// TIA Portal project "LabKlipovi" (V14)

(* hardware
DEVICE "S71500/ET200MP station_1"  S7-1500 station
   slot 0: "Rail_0"  Rack  6ES7 590-1***0-0AA0
   slot 1: "PLC_1"  CPU 1511-1 PN  6ES7 511-1AK00-0AB0  V1.0
      slot 3: "CPU display_1"  6ES7591-1XA00-0AA0
   slot 2: "DI 16x24VDC HF_1"  DI 16x24VDC HF  6ES7 521-1BH00-0AB0  V1.0
   slot 3: "DQ 16x24VDC/0.5A ST_1"  DQ 16x24VDC/0.5A ST  6ES7 522-1BH00-0AB0  V1.0
   slot 4: "AI 8xU/I/RTD/TC ST_1"  AI 8xU/I/RTD/TC ST  6ES7 531-7KF00-0AB0  V2.0
*)

// ===== PLC "PLC_1"  CPU 1511-1 PN =====

VAR_GLOBAL   // PLC tag table "Tag table_1"
   "K1L" AT %I0.0 : Bool;
   "K1D" AT %I0.1 : Bool;
   "K2L" AT %I0.2 : Bool;
   "K2D" AT %I0.3 : Bool;
   "K3L" AT %I0.4 : Bool;
   "K3D" AT %I0.5 : Bool;
   "K4L" AT %I0.6 : Bool;
   "K4D" AT %I0.7 : Bool;
   "Komanda_K1L" AT %Q0.0 : Bool;
   "Komanda_K1D" AT %Q0.1 : Bool;
   "Komanda_K2L" AT %Q0.2 : Bool;
   "Komanda_K2D" AT %Q0.3 : Bool;
   "Komanda_K3L" AT %Q0.4 : Bool;
   "Komanda_K4L" AT %Q0.6 : Bool;
   "K1_AN" AT %IW2 : Int;
   "K4_AN" AT %IW4 : Int;
   "Timer_12s" AT %T0 : Timer;
   "Counter_0" AT %C0 : Counter;
   "Timer_9s" AT %T1 : Timer;
   "Crank" AT %M0.0 : Bool;
END_VAR

DATA_BLOCK "Block_1_DB"   // DB1
{ S7_Optimized_Access := 'TRUE' }
VERSION : 0.1
// stored: InstanceOfName Block_1
"Block_1"
BEGIN
END_DATA_BLOCK

FUNCTION_BLOCK "Block_1"   // FB1, GRAPH_PLUS
{ S7_Optimized_Access := 'TRUE' }
VERSION : 0.1
   VAR_INPUT
      OFF_SQ : Bool := false;   // Turn sequence off
      INIT_SQ : Bool := false;   // Set sequence to initial state
      ACK_EF : Bool := false;   // Acknowledge all errors and faults
      S_PREV : Bool := false;   // Output previous step in parameter S_NO
      S_NEXT : Bool := false;   // Indicate next step in parameter S_NO
      SW_AUTO : Bool := false;   // Automatic mode
      SW_TAP : Bool := false;   // Semiautomatic/switch with transition
      SW_TOP : Bool := false;   // Semiautomatic/ignore transition
      SW_MAN : Bool := false;   // Manual mode
      S_SEL : Int := 0;   // Select step to be output to S_NO
      S_ON : Bool := false;   // Activate step indicated in S_NO
      S_OFF : Bool := false;   // Deactivate step indicated S_NO
      T_PUSH : Bool := false;   // Enable transition to switch in semi automatic mode
   END_VAR
   VAR_OUTPUT
      S_NO : Int := 0;   // Step number
      S_MORE : Bool := false;   // More steps are available and can be shown in S_NO
      S_ACTIVE : Bool := false;   // Step indicated in S_NO is active
      ERR_FLT : Bool := false;   // Interlock or supervision group error
      AUTO_ON : Bool := false;   // Automatic mode is active
      TAP_ON : Bool := false;   // Semiautomatic mode/step with transition enabled
      TOP_ON : Bool := false;   // Semiautomatic mode/ignore transition enabled
      MAN_ON : Bool := false;   // Manual mode is active
   END_VAR
   VAR
      HMI_INFO : Array[0..10] of UInt;
      IF_PAR : G7_IfParPlus_V2;
      RT_DATA : G7_RTDataPlus_V2;   // Internal data area
      Trans1 : G7_TransitionPlus_V2;   // Transition structure
      Trans2 : G7_TransitionPlus_V2;   // Transition structure
      Trans3 : G7_TransitionPlus_V2;   // Transition structure
      Trans4 : G7_TransitionPlus_V2;   // Transition structure
      Trans5 : G7_TransitionPlus_V2;   // Transition structure
      Trans7 : G7_TransitionPlus_V2;   // Transition structure
      Trans8 : G7_TransitionPlus_V2;   // Transition structure
      Trans10 : G7_TransitionPlus_V2;   // Transition structure
      Trans11 : G7_TransitionPlus_V2;   // Transition structure
      Trans12 : G7_TransitionPlus_V2;   // Transition structure
      Trans14 : G7_TransitionPlus_V2;   // Transition structure
      Trans15 : G7_TransitionPlus_V2;   // Transition structure
      Trans16 : G7_TransitionPlus_V2;   // Transition structure
      Trans17 : G7_TransitionPlus_V2;   // Transition structure
      Trans18 : G7_TransitionPlus_V2;   // Transition structure
      Trans19 : G7_TransitionPlus_V2;   // Transition structure
      Init : G7_StepPlus_V2;   // Step structure
      Step2 : G7_StepPlus_V2;   // Step structure
      Step3 : G7_StepPlus_V2;   // Step structure
      Step4 : G7_StepPlus_V2;   // Step structure
      Step5 : G7_StepPlus_V2;   // Step structure
      Step7 : G7_StepPlus_V2;   // Step structure
      Step8 : G7_StepPlus_V2;   // Step structure
      Step10 : G7_StepPlus_V2;   // Step structure
      Step11 : G7_StepPlus_V2;   // Step structure
      Step12 : G7_StepPlus_V2;   // Step structure
      Step13 : G7_StepPlus_V2;   // Step structure
      Step14 : G7_StepPlus_V2;   // Step structure
      Step15 : G7_StepPlus_V2;   // Step structure
      Step16 : G7_StepPlus_V2;   // Step structure
      Step17 : G7_StepPlus_V2;   // Step structure
      SINI : Array[0..3] of USInt;
      LSTT : Array[0..15] of USInt;
      ATAJ : Array[0..15] of USInt;
      ATAB : Array[0..15] of USInt;
      PSTT : Array[0..15] of USInt;
      NSTT : Array[0..15] of USInt;
      ASSJ : Array[0..14] of USInt;
      ASSB : Array[0..14] of USInt;
      PTTS : Array[0..14] of USInt;
      NTTS : Array[0..14] of USInt;
      SW_SQTS : Array[0..14] of USInt;
      SWITCH : Array[0..1] of USInt;
      TVX : Array[0..5] of USInt;
      TTX : Array[0..5] of USInt;
      TSX : Array[0..3] of USInt;
      S00X : Array[0..3] of USInt;
      SOFFX : Array[0..3] of USInt;
      SONX : Array[0..3] of USInt;
      SAX : Array[0..3] of USInt;
      SERRX : Array[0..15] of USInt;
      SMX : Array[0..15] of USInt;
      S0X : Array[0..15] of USInt;
      S1X : Array[0..15] of USInt;
      IL_ALARM_INST : Program_Alarm;
      SUP_ALARM_INST : Program_Alarm;
      STEP_TIME_ALARM_INST : Program_Alarm;
      IEC_TIMER_INST : IEC_TIMER;
   END_VAR
   // SINI[0] := 2;
   // LSTT[0] := 255;
   // LSTT[1] := 255;
   // LSTT[2] := 255;
   // LSTT[3] := 255;
   // LSTT[4] := 255;
   // LSTT[5] := 255;
   // ATAJ[1] := 1;
   // ATAJ[2] := 2;
   // ATAJ[3] := 3;
   // ATAJ[4] := 4;
   // ATAJ[5] := 5;
   // ATAB[1] := 1;
   // ATAB[2] := 2;
   // ATAB[3] := 3;
   // ATAB[4] := 4;
   // ATAB[5] := 5;
   // PSTT[1] := 1;
   // PSTT[2] := 2;
   // PSTT[3] := 3;
   // PSTT[4] := 4;
   // PSTT[5] := 5;
   // NSTT[0] := 1;
   // NSTT[1] := 2;
   // NSTT[2] := 3;
   // NSTT[3] := 4;
   // NSTT[4] := 5;
   // NSTT[5] := 6;
   // ASSJ[1] := 1;
   // ASSJ[2] := 2;
   // ASSJ[3] := 3;
   // ASSJ[4] := 4;
   // ASSJ[5] := 5;
   // ASSB[1] := 1;
   // ASSB[2] := 2;
   // ASSB[3] := 3;
   // ASSB[4] := 4;
   // ASSB[5] := 7;
   // PTTS[0] := 255;
   // PTTS[2] := 1;
   // PTTS[3] := 2;
   // PTTS[4] := 3;
   // PTTS[5] := 4;
   // NTTS[1] := 1;
   // NTTS[2] := 2;
   // NTTS[3] := 3;
   // NTTS[4] := 4;
   // NTTS[5] := 5;
   // TVX[0] := 16#1;
   // TTX[0] := 16#1;
   // TSX[0] := 16#1;
   // S00X[0] := 16#1;
   // SOFFX[0] := 16#1;
   // SONX[0] := 16#1;
   // SAX[0] := 16#1;
   // SERRX[0] := 16#1;
   // SMX[0] := 16#1;
   // S0X[0] := 16#1;
   // S1X[0] := 16#1;
   // NTTS[8] := 8;
   // PTTS[8] := 7;
   // ASSB[8] := 8;
   // SW_SQTS[8] := 2;
   // ASSJ[8] := 8;
   // SINI[2] := 255;
   // SINI[3] := 255;
   // LSTT[6] := 5;
   // LSTT[7] := 255;
   // NSTT[8] := 9;
   // ATAJ[6] := 6;
   // ATAJ[7] := 7;
   // PSTT[8] := 8;
   // ATAB[6] := 6;
   // ATAB[7] := 7;
   // ATAB[8] := 8;
   // PSTT[6] := 6;
   // PSTT[7] := 7;
   // ATAJ[8] := 8;
   // NSTT[6] := 5;
   // NSTT[7] := 8;
   // LSTT[8] := 255;
   // ASSJ[6] := 6;
   // ASSJ[7] := 7;
   // ASSB[6] := 6;
   // ASSB[7] := 5;
   // PTTS[6] := 5;
   // PTTS[7] := 4;
   // NTTS[6] := 6;
   // NTTS[7] := 7;
   // SW_SQTS[5] := 1;
   // SW_SQTS[6] := 1;
   // SW_SQTS[7] := 2;
   // SWITCH[0] := 192;
   // LSTT[11] := 255;
   // LSTT[9] := 255;
   // LSTT[10] := 3;
   // ATAJ[9] := 9;
   // ATAJ[10] := 10;
   // ATAB[9] := 10;
   // ATAB[10] := 9;
   // PSTT[9] := 10;
   // PSTT[10] := 10;
   // NSTT[9] := 11;
   // NSTT[10] := 3;
   // ASSJ[9] := 9;
   // ASSB[9] := 9;
   // PTTS[9] := 8;
   // NTTS[9] := 11;
   // SW_SQTS[9] := 2;
   // ATAJ[11] := 11;
   // ATAB[11] := 11;
   // PSTT[11] := 9;
   // NSTT[11] := 10;
   // ASSJ[10] := 10;
   // ASSB[10] := 10;
   // PTTS[10] := 11;
   // NTTS[10] := 9;
   // SW_SQTS[10] := 2;
   // LSTT[12] := 255;
   // LSTT[13] := 255;
   // LSTT[14] := 255;
   // LSTT[15] := 255;
   // ATAJ[12] := 12;
   // ATAJ[13] := 13;
   // ATAJ[14] := 14;
   // ATAJ[15] := 15;
   // ATAB[12] := 12;
   // ATAB[13] := 13;
   // ATAB[14] := 14;
   // ATAB[15] := 15;
   // PSTT[12] := 11;
   // PSTT[13] := 12;
   // PSTT[14] := 13;
   // PSTT[15] := 14;
   // NSTT[12] := 12;
   // NSTT[13] := 13;
   // NSTT[14] := 14;
   // NSTT[15] := 255;
   // ASSJ[11] := 11;
   // ASSJ[12] := 12;
   // ASSJ[13] := 13;
   // ASSJ[14] := 14;
   // ASSB[11] := 11;
   // ASSB[12] := 12;
   // ASSB[13] := 13;
   // ASSB[14] := 14;
   // PTTS[11] := 9;
   // PTTS[12] := 12;
   // PTTS[13] := 13;
   // PTTS[14] := 14;
   // NTTS[11] := 12;
   // NTTS[12] := 13;
   // NTTS[13] := 14;
   // NTTS[14] := 15;
   // SW_SQTS[11] := 3;
   // SW_SQTS[12] := 3;
   // SW_SQTS[13] := 3;
   // SW_SQTS[14] := 3;
   // SWITCH[1] := 34;
BEGIN
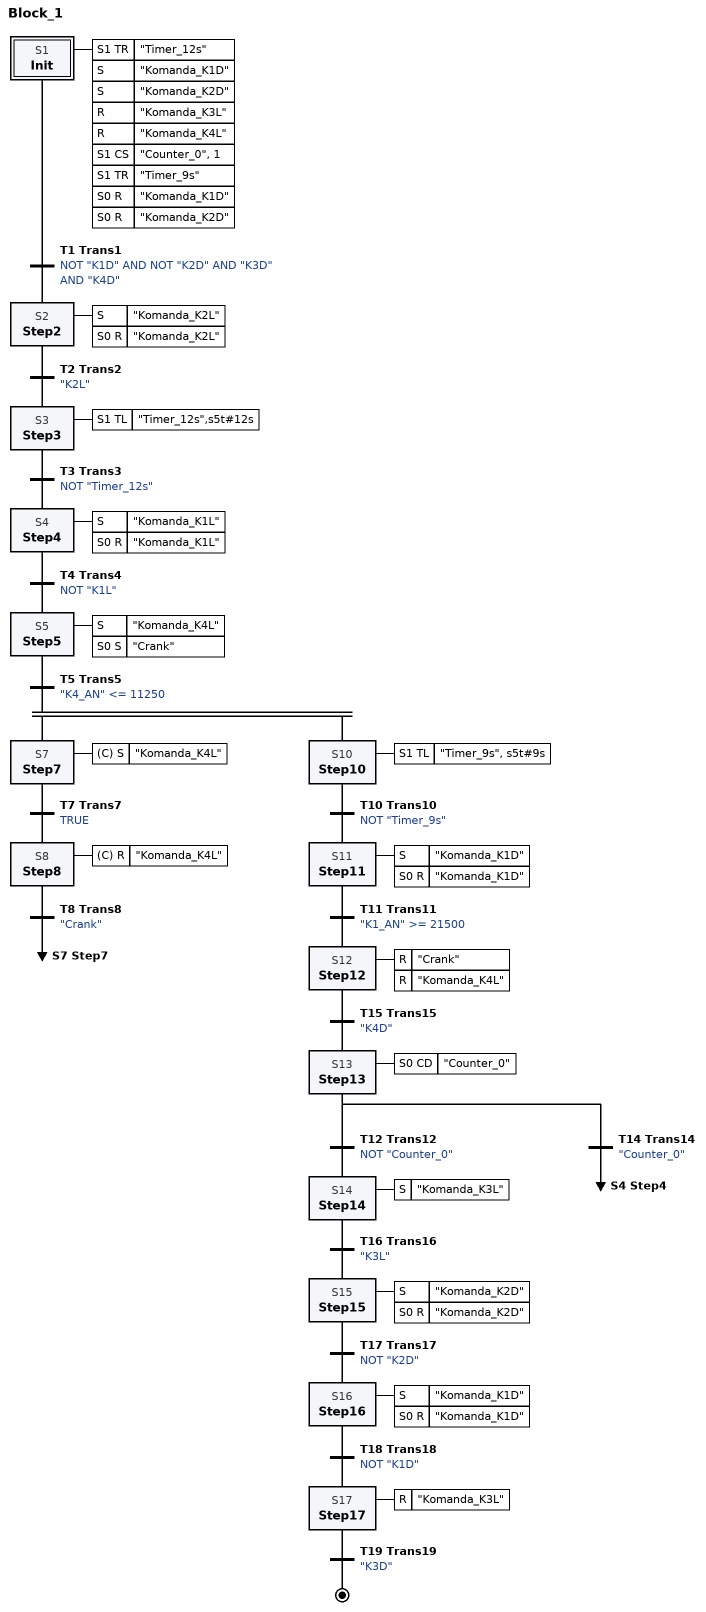
   // sequencer 1
   INITIAL_STEP Init:   // S1, max time T#10S, warning time T#7S
          S1  TR   "Timer_12s"
              S    "Komanda_K1D"
              S    "Komanda_K2D"
              R    "Komanda_K3L"
              R    "Komanda_K4L"
          S1  CS   "Counter_0", 1
          S1  TR   "Timer_9s"
          S0  R    "Komanda_K1D"
          S0  R    "Komanda_K2D"
   END_STEP
   TRANSITION Trans1 FROM Init TO Step2   // T1
      := NOT "K1D" AND NOT "K2D" AND "K3D" AND "K4D";
   END_TRANSITION
   STEP Step2:   // S2, max time T#10S, warning time T#7S
              S    "Komanda_K2L"
          S0  R    "Komanda_K2L"
   END_STEP
   TRANSITION Trans2 FROM Step2 TO Step3   // T2
      := "K2L";
   END_TRANSITION
   STEP Step3:   // S3, max time T#10S, warning time T#7S
          S1  TL   "Timer_12s",s5t#12s
   END_STEP
   TRANSITION Trans3 FROM Step3 TO Step4   // T3
      := NOT "Timer_12s";
   END_TRANSITION
   STEP Step4:   // S4, max time T#10S, warning time T#7S
              S    "Komanda_K1L"
          S0  R    "Komanda_K1L"
   END_STEP
   TRANSITION Trans4 FROM Step4 TO Step5   // T4
      := NOT "K1L";
   END_TRANSITION
   STEP Step5:   // S5, max time T#10S, warning time T#7S
              S    "Komanda_K4L"
          S0  S    "Crank"
   END_STEP
   TRANSITION Trans5 FROM Step5 TO (Step7, Step10)   // T5
      := "K4_AN" <= 11250;
   END_TRANSITION
   STEP Step10:   // S10, max time T#10S, warning time T#7S
          S1  TL   "Timer_9s", s5t#9s
   END_STEP
   TRANSITION Trans10 FROM Step10 TO Step11   // T10
      := NOT "Timer_9s";
   END_TRANSITION
   STEP Step7:   // S7, max time T#10S, warning time T#7S
      interlock C := "K4_AN" >= 11250;
      (C)     S    "Komanda_K4L"
   END_STEP
   TRANSITION Trans7 FROM Step7 TO Step8   // T7
      := TRUE;
   END_TRANSITION
   STEP Step8:   // S8, max time T#10S, warning time T#7S
      interlock C := "K4_AN" <= 11260;
      (C)     R    "Komanda_K4L"
   END_STEP
   TRANSITION Trans8 FROM Step8 TO Step7   // T8, jump
      := "Crank";
   END_TRANSITION
   STEP Step11:   // S11, max time T#10S, warning time T#7S
              S    "Komanda_K1D"
          S0  R    "Komanda_K1D"
   END_STEP
   TRANSITION Trans11 FROM Step11 TO Step12   // T11
      := "K1_AN" >= 21500;
   END_TRANSITION
   STEP Step13:   // S13, max time T#10S, warning time T#7S
          S0  CD   "Counter_0"
   END_STEP
   TRANSITION Trans12 FROM Step13 TO Step14   // T12
      := NOT "Counter_0";
   END_TRANSITION
   TRANSITION Trans14 FROM Step13 TO Step4   // T14, jump
      := "Counter_0";
   END_TRANSITION
   STEP Step12:   // S12, max time T#10S, warning time T#7S
              R    "Crank"
              R    "Komanda_K4L"
   END_STEP
   TRANSITION Trans15 FROM Step12 TO Step13   // T15
      := "K4D";
   END_TRANSITION
   STEP Step14:   // S14, max time T#10S, warning time T#7S
              S    "Komanda_K3L"
   END_STEP
   TRANSITION Trans16 FROM Step14 TO Step15   // T16
      := "K3L";
   END_TRANSITION
   STEP Step15:   // S15, max time T#10S, warning time T#7S
              S    "Komanda_K2D"
          S0  R    "Komanda_K2D"
   END_STEP
   TRANSITION Trans17 FROM Step15 TO Step16   // T17
      := NOT "K2D";
   END_TRANSITION
   STEP Step16:   // S16, max time T#10S, warning time T#7S
              S    "Komanda_K1D"
          S0  R    "Komanda_K1D"
   END_STEP
   TRANSITION Trans18 FROM Step16 TO Step17   // T18
      := NOT "K1D";
   END_TRANSITION
   STEP Step17:   // S17, max time T#10S, warning time T#7S
              R    "Komanda_K3L"
   END_STEP
   TRANSITION Trans19 FROM Step17 TO END   // T19
      := "K3D";
   END_TRANSITION
END_FUNCTION_BLOCK

ORGANIZATION_BLOCK "Main"   // OB1, LAD, ProgramCycle
TITLE = "Main Program Sweep (Cycle)"
{ S7_Optimized_Access := 'TRUE' }
VERSION : 0.1
   VAR_INPUT
      Initial_Call : Bool;   // Initial call of this OB
      Remanence : Bool;   // =True, if remanent data are available
   END_VAR
BEGIN

REGION Network 1
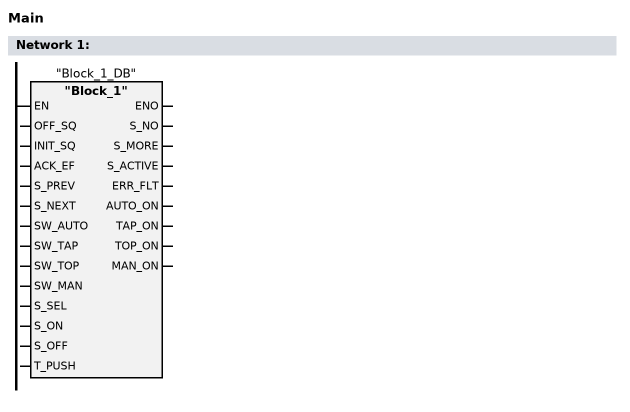
   RUNG wire#powerrail
      "Block_1_DB"(OFF_SQ :=, INIT_SQ :=, ACK_EF :=, S_PREV :=, S_NEXT :=, SW_AUTO :=, SW_TAP :=, SW_TOP :=, SW_MAN :=, S_SEL :=, S_ON :=, S_OFF :=, T_PUSH :=, S_NO =>, S_MORE =>, S_ACTIVE =>, ERR_FLT =>, AUTO_ON =>, TAP_ON =>, TOP_ON =>, MAN_ON =>)
   END_RUNG
   // the same network as SCL:
   "Block_1_DB"();   // "Block_1"
END_REGION
END_ORGANIZATION_BLOCK